// TIA Portal V17 export
// export: Created 2024-03-30T11:13:40.6330757Z, ExportSetting WithDefaults, DisplayName Totally Integrated Automation Portal, DisplayVersion V17, DisplayName TIA Portal Openness, DisplayVersion V17, DisplayName TIA Portal Version Control Interface, DisplayVersion V17, DisplayName STEP 7 Professional, DisplayVersion V17, DisplayName STEP 7 Safety, DisplayVersion V17, DisplayName WinCC Advanced, DisplayVersion V17
DATA_BLOCK "gtyp_MPO"   // DB11
TITLE = Global DB MPO
{ S7_Optimized_Access := 'TRUE' }
AUTHOR : A.Schaefer
VERSION : 0.0
// stored: AutoNumber true, DBAccessibleFromOPCUA true, DBAccessibleFromWebserver true, InstanceOfName typ_MPO, InstanceOfType UDT, IsOnlyStoredInLoadMemory false, IsWriteProtectedInAS false
"typ_MPO"
   // VAR RETAIN
   //    x_Start_Park_Position : Bool;
   //    x_Park_Position_Reached : Bool;
   //    x_Discard_Ready : Bool;
   //    x_MPO_Discards_Accepted : Bool;
   //    x_Error : Bool;
   //    s_ErrorMessage : String := 'No error';
   //    i_PWM_TurnTable : Int := 1000;
   //    i_PWM_Vacuum : Int;
   //    Workpiece : "typ_Workpiece";
   //    Workpiece_Parameters { S7_SetPoint := 'True'} : "typ_Workpiece_Parameters";
   //    History { S7_SetPoint := 'True'} : Array[1..20] of "typ_History";
   // END_VAR
BEGIN
END_DATA_BLOCK
